{ attribute 'Name':='LocalLogMessages-Test' }
{ attribute 'Timeout':='t#5s' }
{ attribute 'Owner':='TestOwner' }
FUNCTION_BLOCK LocalLogMessages_Test_1 EXTENDS FB_TestCaseBase
VAR
	Local		   : LocalLogger;
	Source		   : LogSource;
	Message		   : LogMessage;
	expectedCount  : UDINT;
	actualLogger   : I_Logger;
	expectedLogger : I_Logger	  := Local;
	expectedTime   : T_FILETIME64 := 1234;
	expectedMessage : STRING;
END_VAR

Local.ClearLog();
//Log message
Source.SourceName := 'Test';
Source.Timestamp  := 123456789;
Message.Message	  := 'Message';
Message.Severity  := 12;
Local.LogMessage(Source, Message);
ExpectedMessage := '1601-01-01-00:00:12.345 Test: Message';
AssertMsg(Local.Messages[0] = ExpectedMessage, CONCAT('Expected: ', CONCAT(ExpectedMessage, CONCAT(' Actual: ', Local.Messages[0])))); 

//Test Shift
Source.SourceName := 'Test';
Source.Timestamp  := 123456789;
Message.Message	  := 'Message 2';
Message.Severity  := 12;
Local.LogMessage(Source, Message);
ExpectedMessage := '1601-01-01-00:00:12.345 Test: Message 2';
AssertMsg(Local.Messages[0] = ExpectedMessage, CONCAT('Expected: ', CONCAT(ExpectedMessage, CONCAT(' Actual: ', Local.Messages[0])))); 
ExpectedMessage := '1601-01-01-00:00:12.345 Test: Message';
AssertMsg(Local.Messages[1] = ExpectedMessage, CONCAT('Expected: ', CONCAT(ExpectedMessage, CONCAT(' Actual: ', Local.Messages[1])))); 
Succeeded();

(*Must be implemented if you want to use fastmode*)
METHOD CleanUp : BOOL
//Local.ClearLog();
CleanUp := TRUE;
END_METHOD

END_FUNCTION_BLOCK

(* stored: Version 1.1.0.1, ProductVersion 3.1.4026.18
   POU LocalLogMessages_Test_1: Id {0bc0c4cd-d800-47a4-a75d-872653cea6c2}, SpecialFunc None
   Method Cleanup: Id {e6257f5b-6c80-499e-91de-abe399242abe} *)
